// TIA Portal V18 export
FUNCTION_BLOCK "magnet_"   // FB71, FBD
{ S7_Optimized_Access := 'TRUE' }
VERSION : 0.1
// stored: AutoNumber true, IsIECCheckEnabled false, IsRetainMemResEnabled false, MemoryReserve 100, SetENOAutomatically false, UDAEnableTagReadback false
   VAR_INPUT
      sensor : Bool;
   END_VAR
   VAR_OUTPUT
      y : Bool;
   END_VAR
   VAR
      energize : Bool;
   END_VAR
   VAR RETAIN
      seconds : Real;
   END_VAR
   VAR
      ton { S7_SetPoint := 'True'} : TON_TIME;
      pt_ms : Time;
   END_VAR
BEGIN

REGION Network 1
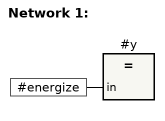
   #y := #energize;
END_REGION

REGION Network 2 (SCL)
   #pt_ms := REAL_TO_DINT(#seconds * 1000.0);
END_REGION
END_FUNCTION_BLOCK
